FUNCTION_BLOCK StackControlLogic
  (* Standard: 61499-2 *)
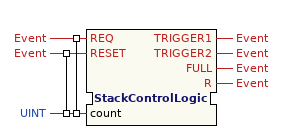
  EVENT_INPUT
    REQ WITH count;
    RESET WITH count;
  END_EVENT
  EVENT_OUTPUT
    TRIGGER1;
    TRIGGER2;
    FULL;
    R;
  END_EVENT
  VAR_INPUT
    count : UINT;
  END_VAR
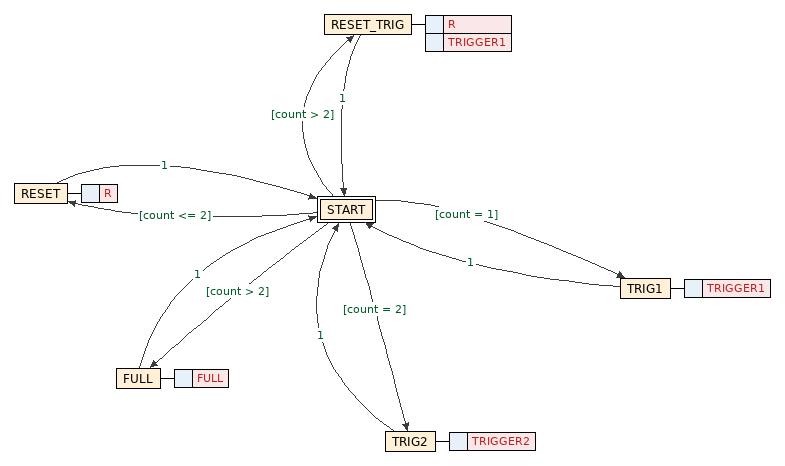
  EC_STATES
    START;
    TRIG1 : -> TRIGGER1;
    TRIG2 : -> TRIGGER2;
    FULL : -> FULL;
    RESET : -> R;
    RESET_TRIG : -> R, -> TRIGGER1;
  END_STATES
  EC_TRANSITIONS
    START TO TRIG1 := [count = 1];
    START TO TRIG2 := [count = 2];
    TRIG2 TO START := 1;
    START TO FULL := [count > 2];
    FULL TO START := 1;
    TRIG1 TO START := 1;
    START TO RESET := [count <= 2];
    RESET TO START := 1;
    START TO RESET_TRIG := [count > 2];
    RESET_TRIG TO START := 1;
  END_TRANSITIONS
END_FUNCTION_BLOCK
